TYPE MB_MAP_VARS_ENUM :
(
	Plant_S_nom:= 0,
	Plant_V_nom:= 1,
	Plant_f_nom:= 2,
	N_converters:= 20,
	nN_converters:= 21,
	Control_conv_0:= 22,
	Control_conv_1:= 23,
	Control_conv_2:= 24,
	Control_conv_3:= 25,
	Control_conv_4:= 26,
	Control_conv_5:= 27,
	Control_conv_6:= 28,
	Control_conv_7:= 29,
	Control_conv_8:= 30,
	Control_conv_9:= 31,
	Control_conv_10:= 32,
	Control_conv_11:= 33,
	Control_conv_12:= 34,
	Control_conv_13:= 35,
	Control_conv_14:= 36,
	Control_conv_15:= 37,
	Control_conv_16:= 38,
	Control_conv_17:= 39,
	Control_conv_18:= 40,
	Control_conv_19:= 41,
	Control_conv_20:= 42,
	Control_conv_21:= 43,
	Control_conv_22:= 44,
	Control_conv_23:= 45,
	Control_conv_24:= 46,
	Control_conv_25:= 47,
	P_loop:= 300,
	P_refence:= 301,
	P_feedback:= 302,
	P_output:= 303,
	P_kp:= 304,
	P_kp_min:= 305,
	P_ti:= 306,
	P_high:= 307,
	P_low:= 308,
	P_invert:= 309,
	P_safety:= 310,
	Q_loop:= 500,
	Q_refence:= 501,
	Q_feedback:= 502,
	Q_output:= 503,
	Q_kp:= 504,
	Q_kp_min:= 505,
	Q_ti:= 506,
	Q_high:= 507,
	Q_low:= 508,
	Q_invert:= 509,
	Q_safety:= 510,
	Ramp_enable:= 511,
	Time_span:= 512,
	R_up_value:= 513,
	R_down_value:= 514,
	R_units:= 515,
	P_L1_kW:= 1000,
	P_L2_kW:= 1002,
	P_L3_kW:= 1004,
	Q_L1_kVAr:= 1006,
	Q_L2_kVAr:= 1008,
	Q_L3_kVAr:= 1010,
	S_L1_kVA:= 1012,
	S_L2_kVA:= 1014,
	S_L3_kVA:= 1016,
	cos_phi_L1:= 1018,
	cos_phi_L2:= 1020,
	cos_phi_L3:= 1022,
	V_L1N_Volt:= 1024,
	V_L2N_Volt:= 1026,
	V_L3N_Volt:= 1028,
	P_tot_kW:= 1030,
	Q_tot_kVAr:= 1032,
	S_tot_kVA:= 1034,
	Freq_Hz:= 1036,
	cos_phi:= 1038,
	V_L1L2_Volt:= 1040,
	V_L2L3_Volt:= 1042,
	V_L3L1_Volt:= 1044,
	I_L1_angle:= 1046,
	I_L2_angle:= 1048,
	I_L3_angle:= 1050,
	V_L1L2_angle:= 1052,
	V_L1L3_angle:= 1054,
	V_phase_avg_Volt:= 1080,
	V_line_avg_Volt:= 1082,
	P_L1_pu:= 1084,
	P_L2_pu:= 1086,
	P_L3_pu:= 1088,
	Q_L1_pu:= 1090,
	Q_L2_pu:= 1092,
	Q_L3_pu:= 1094,
	S_L1_pu:= 1096,
	S_L2_pu:= 1098,
	S_L3_pu:= 1100,
	P_tot_pu:= 1102,
	Q_tot_pu:= 1104,
	S_tot_pu:= 1106,
	V_phase_avg_pu:= 1108,
	V_line_avg_pu:= 1110,
	Active_er_pos_kWh:= 1200,
	Active_er_neg_kWh:= 1204,
	Active_er_tot_kWh:= 1208,
	React_er_pos_kVArh:= 1212,
	React_er_neg_kVArh:= 1216,
	React_er_tot_kVArh:= 1220,
	Energies_reset:= 1224,
	Meter_status:= 1130,
	Lost_comms_enable:= 1131	
);
END_TYPE

(* stored: Version 1.1.0.1, ProductVersion 3.1.4024.11
   EnumerationTextList MB_MAP_VARS_ENUM: Id {7ec9e1d6-220f-422b-9ddc-4aed3e74df3f} *)
